DATA_BLOCK "ST10_PMCountCycleTime"
{ S7_Optimized_Access := 'FALSE' }
VERSION : 0.1
NON_RETAIN
// ATTRIBUTES
// AUTO_NUMBER = False
// BLOCK_NUMBER = 1061
// END_ATTRIBUTES
   STRUCT
      PM { S7_SetPoint := 'False'} : Array[1..30] of "RCS_CountCycleTime_V1";
      PM_Num : Int;
   END_STRUCT;


BEGIN

END_DATA_BLOCK

